# EPICS autosave request: ipApp/Db/PTC10_settings.req
$(P)$(T):outputEnable
$(P)$(T):outputEnable_RBV.SCAN
